{attribute 'qualified_only'}
{attribute 'strict'}
TYPE E_RFIDState :
(
	Idle			:= 0,
	Clearing		:= 1,
	Reading			:= 2,
	Completing		:= 3
);
END_TYPE

(* stored: Version 1.1.0.1, ProductVersion 3.1.4024.4
   DUT E_RFIDState: Id {9d959571-646c-4bbc-8a64-3e2f629779ae} *)
